// TwinCAT 3 PLC project SimulationPLC
// ProgramVersion: 3.1.4022.7
// libraries:
//   Tc2_Standard, * (Beckhoff Automation GmbH)
//   Tc2_System, * (Beckhoff Automation GmbH)
//   Tc3_Module, * (Beckhoff Automation GmbH)
// project tree:
//   / GlobalTextList.TcGTLO, PlcTask.TcTTO, VisualizationManager.TcVMO (not stored), VISU_TASK.TcTTO
//   GVLs/Communication/ DataExchange.TcGVL
//   POUs/Common/ FB_Actuator.TcPOU, FB_Conveyor.TcPOU, FB_SquareWave.TcPOU, FB_ToggleSwitch.TcPOU
//   POUs/ MAIN.TcPOU
//   Visualization/ V_Main.TcVIS
// real-time tasks:
//   TASK PlcTask: cycle T#10ms, priority 20, ADS port 350
//   TASK VISU_TASK: cycle T#200000us, priority 30, ADS port 351

CONFIGURATION SimulationPLC
    RESOURCE PLC ON TwinCAT3
        TASK PlcTask(INTERVAL := T#10ms, PRIORITY := 20);
        TASK VISU_TASK(INTERVAL := T#200000us, PRIORITY := 30);
        PROGRAM MAIN WITH PlcTask : MAIN;
        PROGRAM VisuElems_Visu_Prg WITH VISU_TASK : VisuElems.Visu_Prg;
    END_RESOURCE
END_CONFIGURATION

// ---- GVLs/Communication/DataExchange.TcGVL
{attribute 'qualified_only'}
VAR_GLOBAL
	bVar1			: BOOL;
	iVar1			: DINT;
	button1 		: BOOL;
	status1 		: BOOL;
	
	sensor1 		: BOOL;
	motor1			: BOOL;

	sensor2			: BOOL;	
	motor2			: BOOL;

	sensor3			: BOOL;	
	motor3			: BOOL;
	
	sensor4			: BOOL;	
	motor4			: BOOL;
	
	extend  		: BOOL;
	retract			: BOOL;	
	extended		: BOOL;
	retracted		: BOOL;
	
	pusherFwd		: BOOL;
	pusherBwd		: BOOL;
	
	pusherExtended	: BOOL;
	pusherRetracted	: BOOL;
	
	DAC_Sens_Work	: BOOL;
	DAC_Sens_Home	: BOOL;
	
	DAC_Coil_Work	: BOOL;
	DAC_Coil_Home	: BOOL;
	
	
	
END_VAR

// ---- POUs/MAIN.TcPOU
PROGRAM MAIN
VAR
	fbWave			: FB_SquareWave;
	fbToggle		: FB_ToggleSwitch;
	
	fbInletConv		: FB_Conveyor;
	fbConveyor		: FB_Conveyor;
	fbConveyor_2	: FB_Conveyor;
	fbConveyor_3	: FB_Conveyor;
	
	fbActuator		: FB_Actuator;
	
	iPulseLength	: DINT;
	
	testInt			: REAL;
	sequenceStep	: INT;
	
	handover		: BOOL;
	
	GoToWork		: BOOL;
	GoToHome		: BOOL;
	InWork			: BOOL;
	InHome			: BOOL;
	
END_VAR


iPulseLength := DataExchange.iVar1;	// helper variable - pulse length in ms

fbWave(PulseLength := iPulseLength);	// instance of FB_SquareWave

DataExchange.bVar1 := fbWave.Value;

fbToggle(
	switch := DataExchange.button1,
	status => DataExchange.status1);

fbActuator(
	Sensor_Work := DataExchange.DAC_Sens_Work,
	Sensor_Home := DataExchange.DAC_Sens_Home,
	GoToPos_Work := GoToWork,
	GoToPos_Home := GoToHome,
	ToPos_Work => DataExchange.DAC_Coil_Work,
	ToPos_Home => DataExchange.DAC_Coil_Home,
	InPos_Work => InWork,
	InPos_Home => InHome);
	
fbInletConv(
	Occupied := 	DataExchange.sensor1,
	Handover := 	handover AND fbConveyor.Taking,
	Takeover :=		fbConveyor_3.Giving OR sequenceStep = 10,
	EnableMotor =>	DataExchange.motor1
);
	
fbConveyor(
	Occupied := 	DataExchange.sensor2,
	Handover := 	fbConveyor_2.Taking,
	Takeover :=		fbInletConv.Giving,
	EnableMotor =>	DataExchange.motor2
);

fbConveyor_2(
	Occupied := 	DataExchange.sensor3,
	Handover := 	fbConveyor_3.Taking,
	Takeover :=		fbConveyor.Giving,
	EnableMotor =>	DataExchange.motor3
);

fbConveyor_3(
	Occupied := 	DataExchange.sensor4,
	Handover := 	fbInletConv.Taking,
	Takeover :=		fbConveyor_2.Giving,
	EnableMotor =>	DataExchange.motor4
);



CASE sequenceStep OF
	0: 
		handover := FALSE;
		IF DataExchange.pusherRetracted OR NOT DataExchange.pusherExtended THEN
			IF DataExchange.retracted OR NOT DataExchange.extended THEN
				DataExchange.extend := TRUE;
				DataExchange.retract := FALSE;				
			END_IF
		ELSE
			DataExchange.pusherBwd := TRUE;
			DataExchange.pusherFwd := FALSE;
		END_IF
		
		IF (DataExchange.pusherRetracted OR NOT DataExchange.pusherExtended) AND DataExchange.extended THEN
			sequenceStep := 10;
		END_IF
	10:
		IF DataExchange.sensor1 AND NOT DataExchange.motor1 THEN
			DataExchange.pusherFwd := TRUE;
			DataExchange.pusherBwd := FALSE;
		END_IF	
		IF DataExchange.pusherExtended THEN
			sequenceStep := 20;
		END_IF
	20: 
		DataExchange.pusherBwd := TRUE;
		DataExchange.pusherFwd := FALSE;
		IF DataExchange.pusherRetracted THEN
			sequenceStep := 30;
		END_IF
	30: 
		DataExchange.extend := FALSE;
		DataExchange.retract := TRUE;	
		IF DataExchange.retracted THEN
			handover := TRUE;
			sequenceStep := 40;
		END_IF
	40: 
		IF NOT DataExchange.sensor1 THEN
			handover := FALSE;
			sequenceStep := 0;
		END_IF
END_CASE

END_PROGRAM

// ---- POUs/Common/FB_SquareWave.TcPOU
FUNCTION_BLOCK FB_SquareWave
VAR_INPUT
	PulseLength	: DINT;		// Pulse length in [ms]
END_VAR
VAR_OUTPUT
	Value		: BOOL;
END_VAR
VAR
	Flasher_On	: TON;
	Edge		: BOOL;
END_VAR


Flasher_On(IN := NOT Flasher_On.Q, PT := DINT_TO_TIME(PulseLength));

IF Flasher_On.Q THEN
	Flasher_On(IN := FALSE);
	Edge := TRUE;
END_IF

IF Edge AND Value THEN
	Value := FALSE;
	Edge := FALSE;
ELSIF Edge AND NOT Value THEN
	Value := TRUE;
	Edge := FALSE;
END_IF

END_FUNCTION_BLOCK

// ---- POUs/Common/FB_ToggleSwitch.TcPOU
FUNCTION_BLOCK FB_ToggleSwitch
VAR_INPUT
	switch : BOOL;
END_VAR
VAR_OUTPUT
	status : BOOL;
END_VAR
VAR
	pEdge : BOOL;
END_VAR


IF switch AND NOT pEdge THEN
	pEdge := TRUE;
	IF NOT status THEN
		status := TRUE;
	ELSE
		status := FALSE;
	END_IF
END_IF

pEdge := switch;

END_FUNCTION_BLOCK

// ---- POUs/Common/FB_Conveyor.TcPOU
FUNCTION_BLOCK FB_Conveyor
VAR_INPUT
	Occupied	: BOOL;
	Takeover	: BOOL;
	Handover	: BOOL;
END_VAR
VAR_OUTPUT
	EnableMotor	: BOOL;
	Taking		: BOOL;
	Giving		: BOOL;
END_VAR
VAR
	transportState	: INT;
END_VAR


CASE transportState OF
	0:
	// Init
		Taking 		:= FALSE;
		Giving 		:= FALSE;
		EnableMotor := FALSE;
		transportState := 10;
	10:
	// Takeover or handover
		IF NOT Occupied THEN
			Taking 			:= TRUE;
			Giving 			:= FALSE;
			transportState 	:= 20;	
		ELSE
			Taking 			:= FALSE;
			Giving 			:= TRUE;
			transportState 	:= 200;
		END_IF
	20:
	// Takeover start
		IF Takeover THEN
			EnableMotor 	:= TRUE;
			transportState 	:= 21;
		END_IF		
	21:
	// Occupied
		IF Occupied THEN
			EnableMotor 	:= FALSE;
			Taking			:= FALSE;
			transportState 	:= 10;	
		END_IF		
	200:
	// Handover start
		IF Handover THEN
			Giving 			:= TRUE;
			EnableMotor 	:= TRUE;
			transportState 	:= 210;	
		END_IF
	210:
	// Handover completed
		IF NOT Occupied AND NOT Handover THEN
			EnableMotor		:= FALSE;
			Giving			:= FALSE;
			transportState 	:= 10;	
		END_IF
END_CASE

END_FUNCTION_BLOCK

// ---- POUs/Common/FB_Actuator.TcPOU
FUNCTION_BLOCK FB_Actuator
VAR_INPUT	
	Sensor_Work		: BOOL;
	Sensor_Home		: BOOL;	
	GoToPos_Work	: BOOL;
	GoToPos_Home	: BOOL;	
END_VAR
VAR_OUTPUT	
	ToPos_Work		: BOOL;
	ToPos_Home		: BOOL;	
	InPos_Work		: BOOL;
	InPos_Home		: BOOL;		
END_VAR
VAR
	Moving			: BOOL;
END_VAR


// Reset Outputs
ToPos_Work	:= FALSE;
ToPos_Home	:= FALSE;

// Movement initiated
IF (Sensor_Home AND GoToPos_Work) OR
	(Sensor_Work AND GoToPos_Home) OR 
	(NOT Sensor_Home AND NOT Sensor_Work AND (GoToPos_Work OR GoToPos_Home))THEN
	Moving := TRUE;
END_IF

// Position reached
InPos_Home := Sensor_Home AND NOT Sensor_Work;
InPos_Work := Sensor_Work AND NOT Sensor_Home;

IF (InPos_Home AND GoToPos_Home) THEN
	Moving := FALSE;
END_IF

IF (InPos_Work AND GoToPos_Work) THEN
	Moving := FALSE;
END_IF

// Trigger outputs when valid move initiated
IF Moving AND GoToPos_Work THEN
	ToPos_Work := TRUE;
END_IF

IF Moving AND GoToPos_Home THEN
	ToPos_Home := TRUE;
END_IF

END_FUNCTION_BLOCK

// ---- GlobalTextList.TcGTLO
TEXTLIST GlobalTextList
  689 = '%s'
  61 = 'Enable motor'
  913 = 'Impulse Length'
  18 = 'Sensor'
  632 = 'Square Wave'
END_TEXTLIST

// ---- Visualization/V_Main.TcVIS
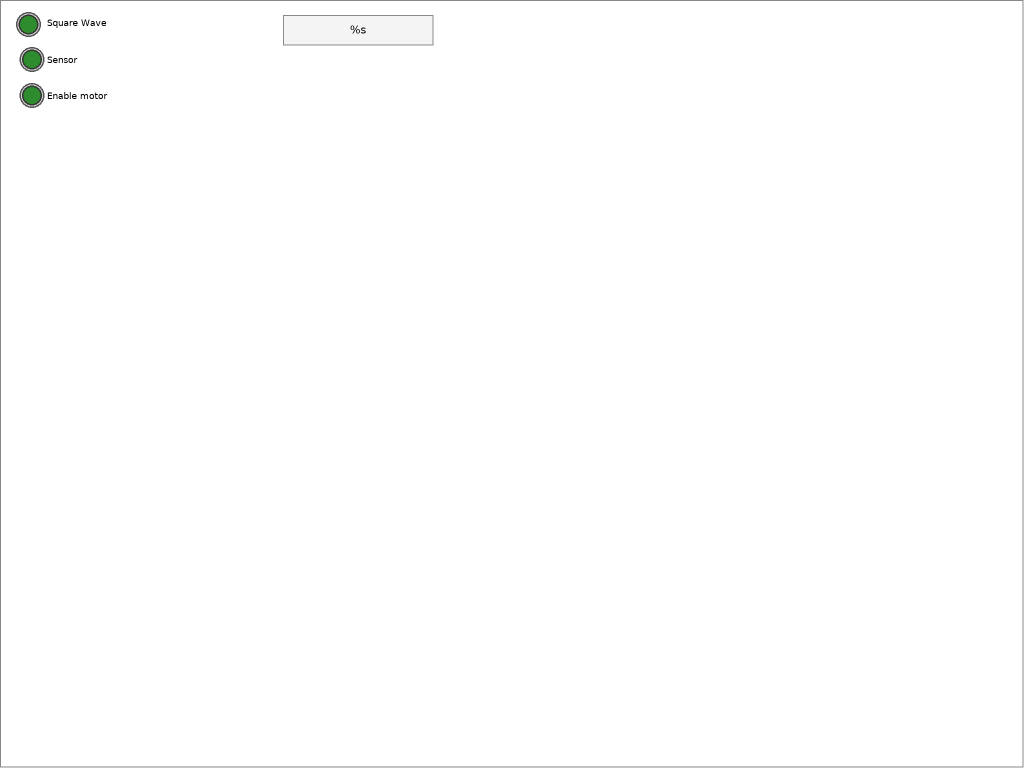
VISUALIZATION V_Main  // 1024x768
    Lamp1 (13,10 31x29), variable: DataExchange.bVar1, style: Lamp-Lamp1-Green
    Lamp1 (13,45 38x29), variable: DataExchange.sensor1, style: Lamp-Lamp1-Green
    Label (44,8 150x30), "Square Wave"
    Label (44,45 150x30), "Sensor"
    Lamp1 (13,81 38x29), variable: DataExchange.motor1, style: Lamp-Lamp1-Green
    Label (44,81 150x30), "Enable motor"
    Scrollbar (283,15 150x30), "%s", text variable: DataExchange.iVar1
        p1057716461: DataExchange.iVar1
END_VISUALIZATION
